TYPE M3GotoKnownPositionArgs :
STRUCT
	///Name of the position (must be configured in M3Config.knownPositions!)
	name: STRING;
END_STRUCT
END_TYPE

(* stored: Version 1.1.0.1, ProductVersion 3.1.4019.2
   DUT M3GotoKnownPositionArgs: Id {842bcfb0-7a5d-4ca7-9745-9b82542030d0} *)
